// TIA Portal V17 export
// export: Created 2023-04-04T13:27:33.6778976Z, ExportSetting WithDefaults, DisplayName Totally Integrated Automation Portal, DisplayVersion V17, DisplayName TIA Portal Openness, DisplayVersion V17, DisplayName TIA Portal Version Control Interface, DisplayVersion V17, DisplayName STEP 7 Professional, DisplayVersion V17, DisplayName STEP 7 Safety, DisplayVersion V17, DisplayName WinCC Advanced, DisplayVersion V17
TYPE "typ_SLD"
// stored: IsFailsafeCompliant false
   STRUCT
      x_Error : Bool;
      i_CounterValue_Blue : Int := 8;
      i_CounterValue_White : Int := 2;
      i_CounterValue_Red : Int := 4;
      i_Counter_Actual : Int;
      w_Threshold_White_Red : Word;
      w_Threshold_Red_Blue : Word;
      Workpiece : "typ_Workpiece";
      History { S7_SetPoint := 'True'} : Array[1..20] of "typ_History";
   END_STRUCT;
END_TYPE
